Omron CX-Programmer project NewProject (CX-Programmer 9.54)

# PLC NewPLC1: CJ1M CPU11

## Global symbols (name address type ; comment)
TimerExample Timer

## Program NewProgram1 (cyclic task 0)

### Section Section1

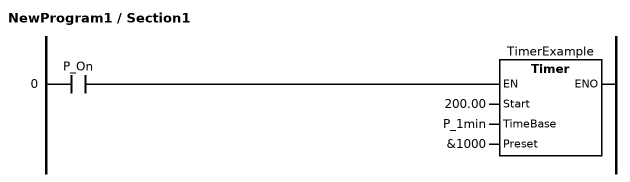
; rung 0
LD P_On
CALL TimerExample : Timer (Start := 200.00, TimeBase := P_1min, Preset := &1000)

### Section END
; rung 0
END(001)

## Function block Timer
VAR_INPUT
  Start : BOOL;
  TimeBase : BOOL;
  Preset : INT;
END_VAR
VAR_OUTPUT
  Running : BOOL;
  Done : BOOL;
  Remaining : INT;
END_VAR
VAR
  TimeBaseOs : BOOL;
  TimeBaseOsAux : BOOL;
  CurrentInternal : INT;
END_VAR
(*TimeBase Oneshot*)
If TimeBase=true then
	If not TimeBaseOsAux then TimeBaseOs:=true;
	Else TimeBaseOs:=false;
	End_if;
End_if;

(*TimeBase Oneshot Aux*)
If TimeBase=true then TimeBaseOsAux:=true;
	Else TimeBaseOsAux:=false;
End_if;

(*Start - increment timer*)
If Start and TimeBaseOs and not Done  then
	CurrentInternal:=CurrentInternal+1;
End_if;

(*Start off, reset timer*)
If not Start then CurrentInternal:=0;
End_if;

(*Test for counter done*)
If CurrentInternal>=Preset then Done:=true;
	else Done:=false;
End_If;

(*Provide Timing output*)
If Start and not Done then Running:=true;
	else Running:=false;
End_if;

(*Ouput remaining time*)
Remaining:=Preset-CurrentInternal;